Staubli VAL3: _WaitAuto.pgx

public program _WaitAuto()
// Wait here until the machine is prepared to be started
begin
  // Enable Robot Off function........................................................
  bRobotOffAllow=true
  //
  //!change 18.06.05, vdg: Prime area test
  call primeAreaTest()
  //
  // ignore messages if in dry run mode
  if data:setDryRun==false
    call status:setEnabled(WAIT_IMM_AUTO,true)
  endIf
  call status:setEnabled(WAIT_MOULD_OPEN,true)
  call status:setEnabled(WAIT_ROB_ENABLE,true)
  // Stop the robot cycle time timer
  //call stat:stopRobotTime()
  // Wait machine in AUTO.............................................................
  do
    //Robot in position to be able use the Robot Off function.
    if SYS:diMachineInAuto[moduleIndex]==false and SYS:bRobotOffCalled[moduleIndex]
      bAtWaitPosition=true
    endIf
    //!change 08.06.06, vdg: ignore automatic signal in dry run mode
  until ((SYS:diMachineInAuto[moduleIndex]==true or data:setDryRun==true) and SYS:diMouldOpen[moduleIndex]==true and bRobotOff==false)
  //
  // Robot not in position to use Robot Off function..................................
  bAtWaitPosition=false
  //
  call status:setEnabled(WAIT_IMM_AUTO,false)
  call status:setEnabled(WAIT_MOULD_OPEN,false)
  call status:setEnabled(WAIT_ROB_ENABLE,false)
  //
  // Start measuring the take out time
  //call stat:startTakeTime()
  //
  call startAreaTest()
end
